FUNCTION F_Variable_DeviceLink: BOOL

GVL_IO.aDigitalInputIO[1].0:=GVL_IO_GAS_CABINET.DI_01_ResetButton ;
GVL_IO.aDigitalInputIO[1].1:=GVL_IO_GAS_CABINET.DI_01_GasCabinetLampButton ;
GVL_IO.aDigitalInputIO[1].2:=GVL_IO_GAS_CABINET.DI_01_PneumaticPressureSensor ;
GVL_IO.aDigitalInputIO[1].3:=GVL_IO_GAS_CABINET.DI_01_GasCabinetDoorClose ;
GVL_IO.aDigitalInputIO[1].4:=GVL_IO_GAS_CABINET.DI_01_ControlCabinetDoorClose ;
GVL_IO.aDigitalInputIO[1].5:=GVL_IO_GAS_CABINET.DI_01_SMPS_1Alarm ;
GVL_IO.aDigitalInputIO[1].6:=GVL_IO_GAS_CABINET.DI_01_SMPS_2Alarm ;
GVL_IO.aDigitalInputIO[1].7:=GVL_IO_GAS_CABINET.DI_01_SMPS_3Alarm ;

GVL_IO.aDigitalInputIO[2].0:=GVL_IO_GAS_CABINET.DI_02_SMPS_4Alarm ;
GVL_IO.aDigitalInputIO[2].1:=GVL_IO_GAS_CABINET.DI_02_GraphiteHeaterELCB ;
GVL_IO.aDigitalInputIO[2].2:=GVL_IO_GAS_CABINET.DI_02_ThermalBathsELCB ;
GVL_IO.aDigitalInputIO[2].3:=GVL_IO_GAS_CABINET.DI_02_VacuumPumpELCB ;
GVL_IO.aDigitalInputIO[2].4:=GVL_IO_GAS_CABINET.DI_02_LineHeatersELCB ;
GVL_IO.aDigitalInputIO[2].5:=GVL_IO_GAS_CABINET.DI_02_RotationMotorCP ;
GVL_IO.aDigitalInputIO[2].6:=GVL_IO_GAS_CABINET.DI_02_CoverLiftMotorCP ;
GVL_IO.aDigitalInputIO[2].7:=GVL_IO_GAS_CABINET.DI_02_T_VCP ;

GVL_IO.aDigitalInputIO[3].0:=GVL_IO_GAS_CABINET.DI_03_GasDetectorCP ;
GVL_IO.aDigitalInputIO[3].1:=GVL_IO_GAS_CABINET.DI_03_CabinetLampsCP ;
GVL_IO.aDigitalInputIO[3].2:=GVL_IO_GAS_CABINET.DI_03_MFCPowerCP ;
GVL_IO.aDigitalInputIO[3].3:=GVL_IO_GAS_CABINET.DI_03_LineHeater_1CP ;
GVL_IO.aDigitalInputIO[3].4:=GVL_IO_GAS_CABINET.DI_03_LineHeater_2CP ;
GVL_IO.aDigitalInputIO[3].5:=GVL_IO_GAS_CABINET.DI_03_LineHeater_3CP ;
GVL_IO.aDigitalInputIO[3].6:=GVL_IO_GAS_CABINET.DI_03_LineHeater_4CP ;
GVL_IO.aDigitalInputIO[3].7:=GVL_IO_GAS_CABINET.DI_03_LineHeater_5CP ;

GVL_IO.aDigitalInputIO[4].0:=GVL_IO_GAS_CABINET.DI_04_LineHeater_6CP ;
GVL_IO.aDigitalInputIO[4].1:=GVL_IO_GAS_CABINET.DI_04_LineHeater_7CP ;
GVL_IO.aDigitalInputIO[4].2:=GVL_IO_GAS_CABINET.DI_04_LineHeater_8CP ;
GVL_IO.aDigitalInputIO[4].3:=GVL_IO_GAS_CABINET.DI_04_GasDetectorH2 ;
GVL_IO.aDigitalInputIO[4].4:=GVL_IO_GAS_CABINET.DI_04_GasDetectorH2S ;
GVL_IO.aDigitalInputIO[4].5:=GVL_IO_GAS_CABINET.DI_04_GasDetectorH2Se ;
GVL_IO.aDigitalInputIO[4].6:=GVL_IO_GAS_CABINET.DI_04_FireSensor ;
GVL_IO.aDigitalInputIO[4].7:=GVL_IO_GAS_CABINET.DI_04_ExternalScrubberFault ;

GVL_IO.aDigitalInputIO[5].0:=GVL_IO_GAS_CABINET.DI_05_ExternalH2GasCabinetFault ;
GVL_IO.aDigitalInputIO[5].1:=GVL_IO_GAS_CABINET.DI_05_ExternalH2SGasCabinetFault ;
GVL_IO.aDigitalInputIO[5].2:=GVL_IO_GAS_CABINET.DI_05_ExternalH2SeGasCabinetFault ;
GVL_IO.aDigitalInputIO[5].3:=GVL_IO_GAS_CABINET.DI_05_ExternalUserInputAlarm ;
GVL_IO.aDigitalInputIO[5].4:=GVL_IO_GAS_CABINET.DI_05_ThermalBath_1DeviationAlarm ;
GVL_IO.aDigitalInputIO[5].5:=GVL_IO_GAS_CABINET.DI_05_ThermalBath_1CutOffAlarm ;
GVL_IO.aDigitalInputIO[5].6:=GVL_IO_GAS_CABINET.DI_05_ThermalBath_2DeviationAlarm ;
GVL_IO.aDigitalInputIO[5].7:=GVL_IO_GAS_CABINET.DI_05_ThermalBath_2CutOffAlarm ;

GVL_IO.aDigitalInputIO[6].0:=GVL_IO_GAS_CABINET.DI_06_ThermalBath_3DeviationAlarm ;
GVL_IO.aDigitalInputIO[6].1:=GVL_IO_GAS_CABINET.DI_06_ThermalBath_3CutOffAlarm ;
GVL_IO.aDigitalInputIO[6].2:=GVL_IO_GAS_CABINET.DI_06_ThermalBath_4DeviationAlarm ;
GVL_IO.aDigitalInputIO[6].3:=GVL_IO_GAS_CABINET.DI_06_ThermalBath_4CutOffAlarm ;
GVL_IO.aDigitalInputIO[6].4:=GVL_IO_GAS_CABINET.DI_06_Spare_01 ;
GVL_IO.aDigitalInputIO[6].5:=GVL_IO_GAS_CABINET.DI_06_Spare_02 ;
GVL_IO.aDigitalInputIO[6].6:=GVL_IO_GAS_CABINET.DI_06_Spare_03 ;
GVL_IO.aDigitalInputIO[6].7:=GVL_IO_GAS_CABINET.DI_06_Spare_04 ;

GVL_IO.aDigitalInputIO[7].0:=GVL_IO_REACTOR_CABINET.DI_01_MaintenanceModeKey ;
GVL_IO.aDigitalInputIO[7].1:=GVL_IO_REACTOR_CABINET.DI_01_ReactorCabinetLampButton ;
GVL_IO.aDigitalInputIO[7].2:=GVL_IO_REACTOR_CABINET.DI_01_DORVACButton ;
GVL_IO.aDigitalInputIO[7].3:=GVL_IO_REACTOR_CABINET.DI_01_DORATMButton ;
GVL_IO.aDigitalInputIO[7].4:=GVL_IO_REACTOR_CABINET.DI_01_ReactorDoorUpButton ;
GVL_IO.aDigitalInputIO[7].5:=GVL_IO_REACTOR_CABINET.DI_01_ReactorDoorDownButton ;
GVL_IO.aDigitalInputIO[7].6:=GVL_IO_REACTOR_CABINET.DI_01_ClampLock ;
GVL_IO.aDigitalInputIO[7].7:=GVL_IO_REACTOR_CABINET.DI_01_ClampRelease ;

GVL_IO.aDigitalInputIO[8].0:=GVL_IO_REACTOR_CABINET.DI_02_C_WFlowSensor ;
GVL_IO.aDigitalInputIO[8].1:=GVL_IO_REACTOR_CABINET.DI_02_SusceptorRotationMotorFault ;
GVL_IO.aDigitalInputIO[8].2:=GVL_IO_REACTOR_CABINET.DI_02_VacuumPumpFail ;
GVL_IO.aDigitalInputIO[8].3:=GVL_IO_REACTOR_CABINET.DI_02_VacuumPumpWarning ;
GVL_IO.aDigitalInputIO[8].4:=GVL_IO_REACTOR_CABINET.DI_02_VacuumPumpAlarm ;
GVL_IO.aDigitalInputIO[8].5:=GVL_IO_REACTOR_CABINET.DI_02_VacuumPumpRunning ;
GVL_IO.aDigitalInputIO[8].6:=GVL_IO_REACTOR_CABINET.DI_02_VacuumPumpFBRunning ;
GVL_IO.aDigitalInputIO[8].7:=GVL_IO_REACTOR_CABINET.DI_02_ReactorDoorUpLimitSensor ;

GVL_IO.aDigitalInputIO[9].0:=GVL_IO_REACTOR_CABINET.DI_03_ReactorDoorDownLimitSensor ;
GVL_IO.aDigitalInputIO[9].1:=GVL_IO_REACTOR_CABINET.DI_03_CylinderAutoSwitch_Closed ;
GVL_IO.aDigitalInputIO[9].2:=GVL_IO_REACTOR_CABINET.DI_03_CylinderAutoSwitch_Opened ;
GVL_IO.aDigitalInputIO[9].3:=GVL_IO_REACTOR_CABINET.DI_03_ReactorCabinetDoorClose ;
GVL_IO.aDigitalInputIO[9].4:=GVL_IO_REACTOR_CABINET.DI_03_Spare_01 ;
GVL_IO.aDigitalInputIO[9].5:=GVL_IO_REACTOR_CABINET.DI_03_Spare_02 ;
GVL_IO.aDigitalInputIO[9].6:=GVL_IO_REACTOR_CABINET.DI_03_Spare_03 ;
GVL_IO.aDigitalInputIO[9].7:=GVL_IO_REACTOR_CABINET.DI_03_Spare_04 ;


GVL_IO.aDigitalOutputIO[1].0:=GVL_IO_GAS_CABINET.DO_07_SystemPowerOffLock ;
GVL_IO.aDigitalOutputIO[1].1:=GVL_IO_GAS_CABINET.DO_07_ControlCabinetLamp ;
GVL_IO.aDigitalOutputIO[1].2:=GVL_IO_GAS_CABINET.DO_07_GasCabinetLamp ;
GVL_IO.aDigitalOutputIO[1].3:=GVL_IO_GAS_CABINET.DO_07_GraphiteHeaterMC ;
GVL_IO.aDigitalOutputIO[1].4:=GVL_IO_GAS_CABINET.DO_07_ThermalBathsMC ;
GVL_IO.aDigitalOutputIO[1].5:=GVL_IO_GAS_CABINET.DO_07_VacuumPumpMC ;
GVL_IO.aDigitalOutputIO[1].6:=GVL_IO_GAS_CABINET.DO_07_LineHeatersMC ;
GVL_IO.aDigitalOutputIO[1].7:=GVL_IO_GAS_CABINET.DO_07_ResetButtonLamp ;

GVL_IO.aDigitalOutputIO[2].0:=GVL_IO_GAS_CABINET.DO_08_Spare_01 ;
GVL_IO.aDigitalOutputIO[2].1:=GVL_IO_GAS_CABINET.DO_08_Spare_02 ;
GVL_IO.aDigitalOutputIO[2].2:=GVL_IO_GAS_CABINET.DO_08_Spare_03 ;
GVL_IO.aDigitalOutputIO[2].3:=GVL_IO_GAS_CABINET.DO_08_Spare_04 ;
GVL_IO.aDigitalOutputIO[2].4:=GVL_IO_GAS_CABINET.DO_08_Spare_05 ;
GVL_IO.aDigitalOutputIO[2].5:=GVL_IO_GAS_CABINET.DO_08_Spare_06 ;
GVL_IO.aDigitalOutputIO[2].6:=GVL_IO_GAS_CABINET.DO_08_Spare_07 ;
GVL_IO.aDigitalOutputIO[2].7:=GVL_IO_GAS_CABINET.DO_08_Spare_08 ;

GVL_IO.aDigitalOutputIO[3].0:=GVL_IO_REACTOR_CABINET.DO_04_SignalTowerRed ;
GVL_IO.aDigitalOutputIO[3].1:=GVL_IO_REACTOR_CABINET.DO_04_SignalTowerOrange ;
GVL_IO.aDigitalOutputIO[3].2:=GVL_IO_REACTOR_CABINET.DO_04_SignalTowerGreen ;
GVL_IO.aDigitalOutputIO[3].3:=GVL_IO_REACTOR_CABINET.DO_04_SignalTowerBlue ;
GVL_IO.aDigitalOutputIO[3].4:=GVL_IO_REACTOR_CABINET.DO_04_SignalTowerWhite ;
GVL_IO.aDigitalOutputIO[3].5:=GVL_IO_REACTOR_CABINET.DO_04_SignalTowerBuzzer ;
GVL_IO.aDigitalOutputIO[3].6:=GVL_IO_REACTOR_CABINET.DO_04_ReactorCoverUpRelay ;
GVL_IO.aDigitalOutputIO[3].7:=GVL_IO_REACTOR_CABINET.DO_04_ReactorCoverDownRelay ;

GVL_IO.aDigitalOutputIO[4].0:=GVL_IO_REACTOR_CABINET.DO_05_ClampLock ;
GVL_IO.aDigitalOutputIO[4].1:=GVL_IO_REACTOR_CABINET.DO_05_ClampRelease ;
GVL_IO.aDigitalOutputIO[4].2:=GVL_IO_REACTOR_CABINET.DO_05_VacuumPumpStart_Stop ;
GVL_IO.aDigitalOutputIO[4].3:=GVL_IO_REACTOR_CABINET.DO_05_VacuumPumpReset ;
GVL_IO.aDigitalOutputIO[4].4:=GVL_IO_REACTOR_CABINET.DO_05_SusceptorRotationFWD ;
GVL_IO.aDigitalOutputIO[4].5:=GVL_IO_REACTOR_CABINET.DO_05_SusceptorRotationSTOP ;
GVL_IO.aDigitalOutputIO[4].6:=GVL_IO_REACTOR_CABINET.DO_05_SusceptorRotationAL_RST ;
GVL_IO.aDigitalOutputIO[4].7:=GVL_IO_REACTOR_CABINET.DO_05_DORVACButtonLamp ;

GVL_IO.aDigitalOutputIO[5].0:=GVL_IO_REACTOR_CABINET.DO_06_DORATMButtonLamp ;
GVL_IO.aDigitalOutputIO[5].1:=GVL_IO_REACTOR_CABINET.DO_06_ReactorCoverUpButtonLamp ;
GVL_IO.aDigitalOutputIO[5].2:=GVL_IO_REACTOR_CABINET.DO_06_ReactorCoverDownButtonLamp ;
GVL_IO.aDigitalOutputIO[5].3:=GVL_IO_REACTOR_CABINET.DO_06_ClampLockButtonLamp ;
GVL_IO.aDigitalOutputIO[5].4:=GVL_IO_REACTOR_CABINET.DO_06_ClampReleaseButtonLamp ;
GVL_IO.aDigitalOutputIO[5].5:=GVL_IO_REACTOR_CABINET.DO_06_ReactorCabinetLamp ;
GVL_IO.aDigitalOutputIO[5].6:=GVL_IO_REACTOR_CABINET.DO_06_Spare07 ;
GVL_IO.aDigitalOutputIO[5].7:=GVL_IO_REACTOR_CABINET.DO_06_Spare08 ;


GVL_IO.aAnalogInputIO[1]:=GVL_IO_GAS_CABINET.AI_09_M01_ChalcogenRunPV ;
GVL_IO.aAnalogInputIO[2]:=GVL_IO_GAS_CABINET.AI_09_M02_MORunPV ;
GVL_IO.aAnalogInputIO[3]:=GVL_IO_GAS_CABINET.AI_09_M03_H2SeSupplyPV ;
GVL_IO.aAnalogInputIO[4]:=GVL_IO_GAS_CABINET.AI_09_M04_H2SSupplyPV ;
GVL_IO.aAnalogInputIO[5]:=GVL_IO_GAS_CABINET.AI_11_M05_Source_1TMInSupplyPV ;
GVL_IO.aAnalogInputIO[6]:=GVL_IO_GAS_CABINET.AI_11_M06_Source_2TMGaSupplyPV ;
GVL_IO.aAnalogInputIO[7]:=GVL_IO_GAS_CABINET.AI_11_M07_Source_3DMSeSupplyPV ;
GVL_IO.aAnalogInputIO[8]:=GVL_IO_GAS_CABINET.AI_11_M08_Source_4ChalcoSupplyPV ;
GVL_IO.aAnalogInputIO[9]:=GVL_IO_GAS_CABINET.AI_13_M09_LinerPurgePV ;
GVL_IO.aAnalogInputIO[10]:=GVL_IO_GAS_CABINET.AI_13_M10_HeaterPurgePV ;
GVL_IO.aAnalogInputIO[11]:=GVL_IO_GAS_CABINET.AI_13_M11_ChalcogenVentPV ;
GVL_IO.aAnalogInputIO[12]:=GVL_IO_GAS_CABINET.AI_13_M12_MOVentPV ;
GVL_IO.aAnalogInputIO[13]:=GVL_IO_GAS_CABINET.AI_15_E01Source_1TMInPressurePV ;
GVL_IO.aAnalogInputIO[14]:=GVL_IO_GAS_CABINET.AI_15_E02Source_2TMGaPressurePV ;
GVL_IO.aAnalogInputIO[15]:=GVL_IO_GAS_CABINET.AI_15_E03Source_3DMSePressurePV ;
GVL_IO.aAnalogInputIO[16]:=GVL_IO_GAS_CABINET.AI_15_E04Source_4ChalcoPressurePV ;
GVL_IO.aAnalogInputIO[17]:=GVL_IO_GAS_CABINET.DI_18_S01N2SupplyPressPV ;
GVL_IO.aAnalogInputIO[18]:=GVL_IO_GAS_CABINET.DI_18_S02H2SupplyPressPV ;
GVL_IO.aAnalogInputIO[19]:=GVL_IO_GAS_CABINET.DI_18_S03H2SSupplyPressPV ;
GVL_IO.aAnalogInputIO[20]:=GVL_IO_GAS_CABINET.DI_18_S04H2SeSupplyPressPV ;
GVL_IO.aAnalogInputIO[21]:=GVL_IO_REACTOR_CABINET.AI_07_P02_ReactorPressure10TorrPV;
GVL_IO.aAnalogInputIO[22]:=GVL_IO_REACTOR_CABINET.AI_07_P03_ExhaustPressurePV ;
GVL_IO.aAnalogInputIO[23]:=GVL_IO_REACTOR_CABINET.AI_07_S05_DORPressurePV ;
GVL_IO.aAnalogInputIO[24]:=GVL_IO_REACTOR_CABINET.AI_07_Spare_04 ;

GVL_IO.aAnalogInputIO[25]:=GVL_IO_REACTOR_CABINET.AI_08_R01SusceptorRotationPV ;
GVL_IO.aAnalogInputIO[26]:=GVL_IO_REACTOR_CABINET.AI_08_Spare_02 ;
GVL_IO.aAnalogInputIO[27]:=GVL_IO_REACTOR_CABINET.AI_08_Spare_03 ;
GVL_IO.aAnalogInputIO[28]:=GVL_IO_REACTOR_CABINET.AI_08_Spare_04 ;

GVL_IO.aAnalogInputIO[29]:=GVL_IO_REACTOR_CABINET.AI_10_R04S_HCoolingWaterPV ;
GVL_IO.aAnalogInputIO[30]:=GVL_IO_REACTOR_CABINET.AI_10_Spare_02 ;
GVL_IO.aAnalogInputIO[31]:=GVL_IO_REACTOR_CABINET.AI_10_Spare_03 ;
GVL_IO.aAnalogInputIO[32]:=GVL_IO_REACTOR_CABINET.AI_10_Spare_04 ;

GVL_IO.aAnalogInputIO2[1]:=GVL_IO_GAS_CABINET.DI_17_DP1ChalcogenDP ;
GVL_IO.aAnalogInputIO2[2]:=GVL_IO_GAS_CABINET.DI_17_DP2MODP ;

GVL_IO_GAS_CABINET.AO_10_M01_ChalcogenRunSV :=GVL_IO.aAnalogOutputIO[1];
GVL_IO_GAS_CABINET.AO_10_M02_MORunSV :=GVL_IO.aAnalogOutputIO[2];
GVL_IO_GAS_CABINET.AO_10_M03_H2SeSupplySV  := GVL_IO.aAnalogOutputIO[3];
GVL_IO_GAS_CABINET.AO_10_M04_H2SSupplySV :=GVL_IO.aAnalogOutputIO[4];

GVL_IO_GAS_CABINET.AO_12_M05_Source_1TMInSupplySV :=GVL_IO.aAnalogOutputIO[5];
GVL_IO_GAS_CABINET.AO_12_M06_Source_2TMGaSupplySV :=GVL_IO.aAnalogOutputIO[6];
GVL_IO_GAS_CABINET.AO_12_M07_Source_3DMSeSupplySV :=GVL_IO.aAnalogOutputIO[7];
GVL_IO_GAS_CABINET.AO_12_M08_Source_4ChalcoSupplySV :=GVL_IO.aAnalogOutputIO[8];
GVL_IO_GAS_CABINET.AO_14_M09_LinerPurgeSV :=GVL_IO.aAnalogOutputIO[9];
GVL_IO_GAS_CABINET.AO_14_M10_HeaterPurgeSV :=GVL_IO.aAnalogOutputIO[10];
GVL_IO_GAS_CABINET.AO_14_M11_ChalcogenVentSV :=GVL_IO.aAnalogOutputIO[11];
GVL_IO_GAS_CABINET.AO_14_M12_MOVentSV :=GVL_IO.aAnalogOutputIO[12];
GVL_IO_GAS_CABINET.AO_16_E01Source_1TMInPressureSV :=GVL_IO.aAnalogOutputIO[13];
GVL_IO_GAS_CABINET.AO_16_E02Source_2TMGaPressureSV :=GVL_IO.aAnalogOutputIO[14];
GVL_IO_GAS_CABINET.AO_16_E03Source_3DMSePressureSV :=GVL_IO.aAnalogOutputIO[15];
GVL_IO_GAS_CABINET.AO_16_E04Source_4ChalcoPressureSV :=GVL_IO.aAnalogOutputIO[16];

GVL_IO_REACTOR_CABINET.AO_09_P03_ExhaustPressureAM215Input:=GVL_IO.aAnalogOutputIO[17];
GVL_IO_REACTOR_CABINET.AO_09_R01_SusceptorRotationSV:=GVL_IO.aAnalogOutputIO[18];
GVL_IO_REACTOR_CABINET.AO_09_Spare_03:=GVL_IO.aAnalogOutputIO[19];
GVL_IO_REACTOR_CABINET.AO_09_Spare_04 :=GVL_IO.aAnalogOutputIO[20];

END_FUNCTION

(* stored: Version 1.1.0.1, ProductVersion 3.1.4024.15
   POU F_Variable_DeviceLink: Id {aa039e23-7245-4b4f-9453-7c5a8340a52e}, SpecialFunc None *)
